// TIA Portal V17 export
// export: Created 2025-06-25T13:13:12.3552397Z, ExportSetting WithDefaults, DisplayName Totally Integrated Automation Portal, DisplayVersion V17 Update 8, DisplayName TIA Portal Openness, DisplayVersion V17 Update 8, DisplayName TIA Portal Version Control Interface, DisplayVersion V17, DisplayName STEP 7 Professional, DisplayVersion V17 Update 8, DisplayName STEP 7 Safety, DisplayVersion V17 Update 6, DisplayName WinCC Advanced, DisplayVersion V17 Update 8
FUNCTION "DigitalOutputProcessing" : Void   // FC11, FBD
TITLE = Output mapping
{ S7_Optimized_Access := 'TRUE' }
VERSION : 0.1
// stored: AutoNumber true, IsIECCheckEnabled false, SetENOAutomatically false, UDAEnableTagReadback false
   VAR_TEMP
      Spare : Bool;
   END_VAR
BEGIN

REGION Network 1: Emergency Stop output
   // 1 = ok, 0 = emergency stop
   // If emergency stop is not active, or you want to reset the safety relay, output is high.
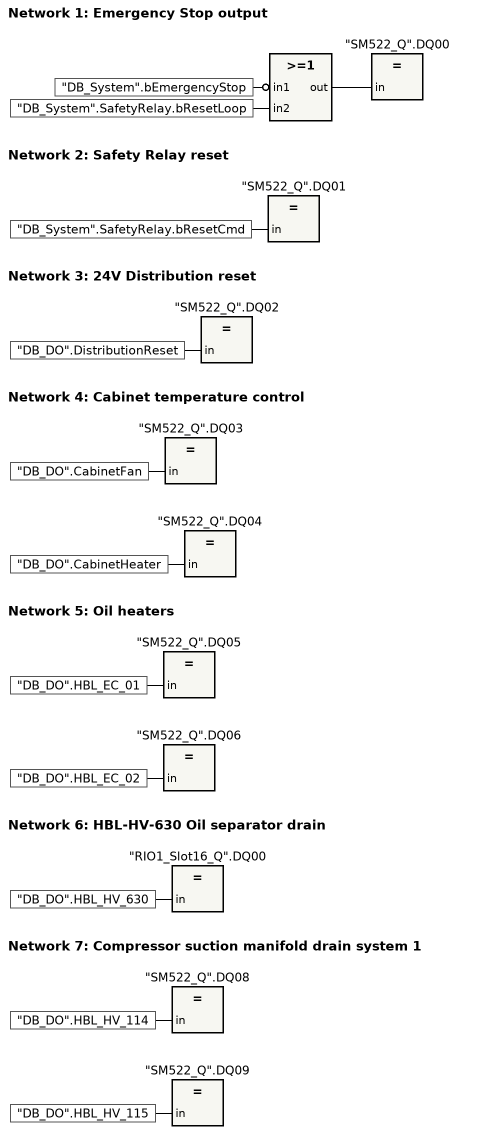
   "SM522_Q".DQ00 := NOT "DB_System".bEmergencyStop OR "DB_System".SafetyRelay.bResetLoop;
END_REGION

REGION Network 2: Safety Relay reset
   "SM522_Q".DQ01 := "DB_System".SafetyRelay.bResetCmd;
END_REGION

REGION Network 3: 24V Distribution reset
   "SM522_Q".DQ02 := "DB_DO".DistributionReset;
END_REGION

REGION Network 4: Cabinet temperature control
   "SM522_Q".DQ03 := "DB_DO".CabinetFan;
   "SM522_Q".DQ04 := "DB_DO".CabinetHeater;
END_REGION

REGION Network 5: Oil heaters
   "SM522_Q".DQ05 := "DB_DO".HBL_EC_01;
   "SM522_Q".DQ06 := "DB_DO".HBL_EC_02;
END_REGION

REGION Network 6: HBL-HV-630 Oil separator drain
   "RIO1_Slot16_Q".DQ00 := "DB_DO".HBL_HV_630;
END_REGION

REGION Network 7: Compressor suction manifold drain system 1
   // Valves directly from suction manifold to sump (optional)
   "SM522_Q".DQ08 := "DB_DO".HBL_HV_114;
   "SM522_Q".DQ09 := "DB_DO".HBL_HV_115;
END_REGION

REGION Network 8: Shaft Seal Cartridge (SSC)
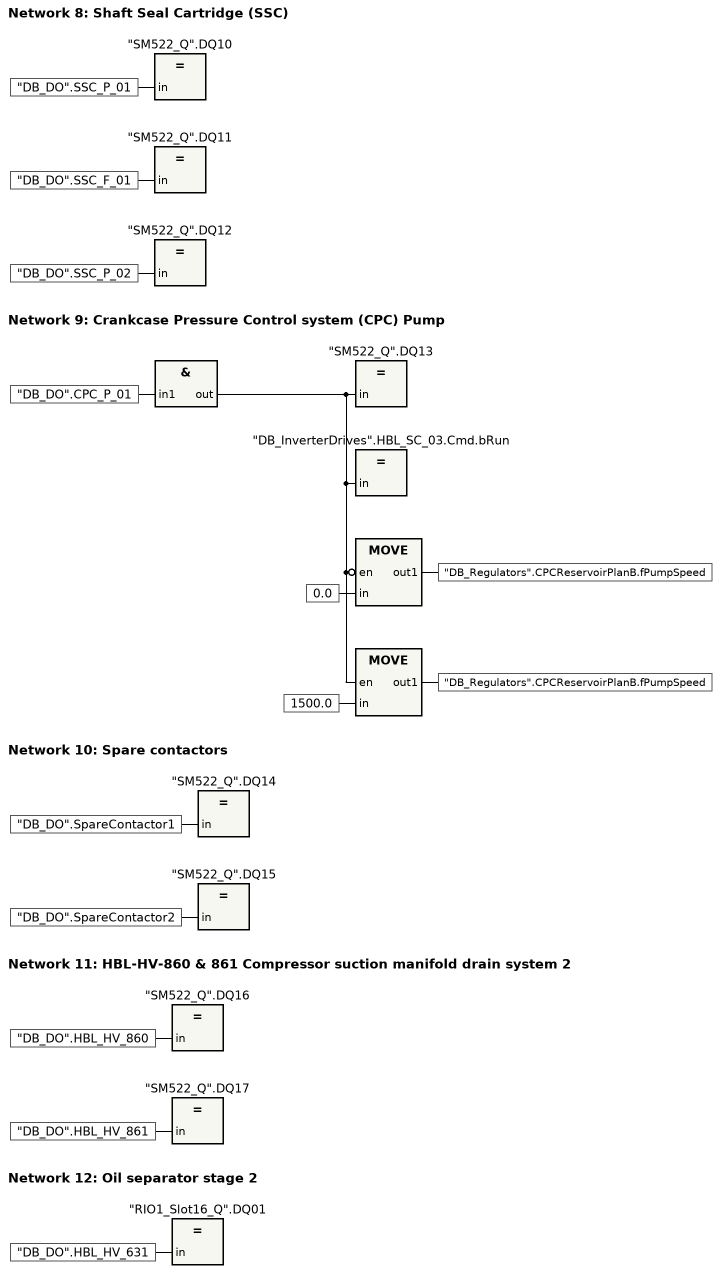
   "SM522_Q".DQ10 := "DB_DO".SSC_P_01;
   "SM522_Q".DQ11 := "DB_DO".SSC_F_01;
   "SM522_Q".DQ12 := "DB_DO".SSC_P_02;
END_REGION

REGION Network 9: Crankcase Pressure Control system (CPC) Pump
   // 10.02.2025 TSS: Normally DQ13, but now an inverter. And this is the ugly hack to make it work until we know how it really should be.
   "SM522_Q".DQ13 := "DB_DO".CPC_P_01;
   "DB_InverterDrives".HBL_SC_03.Cmd.bRun := "DB_DO".CPC_P_01;
   IF NOT "DB_DO".CPC_P_01 THEN "DB_Regulators".CPCReservoirPlanB.fPumpSpeed := 0.0; END_IF;
   IF "DB_DO".CPC_P_01 THEN "DB_Regulators".CPCReservoirPlanB.fPumpSpeed := 1500.0; END_IF;
END_REGION

REGION Network 10: Spare contactors
   "SM522_Q".DQ14 := "DB_DO".SpareContactor1;
   "SM522_Q".DQ15 := "DB_DO".SpareContactor2;
END_REGION

REGION Network 11: HBL-HV-860 & 861 Compressor suction manifold drain system 2
   // Valves to share the CPC system with the Purge controller
   "SM522_Q".DQ16 := "DB_DO".HBL_HV_860;
   "SM522_Q".DQ17 := "DB_DO".HBL_HV_861;
END_REGION

REGION Network 12: Oil separator stage 2
   "RIO1_Slot16_Q".DQ01 := "DB_DO".HBL_HV_631;
END_REGION

REGION Network 13: HBL-HV-640
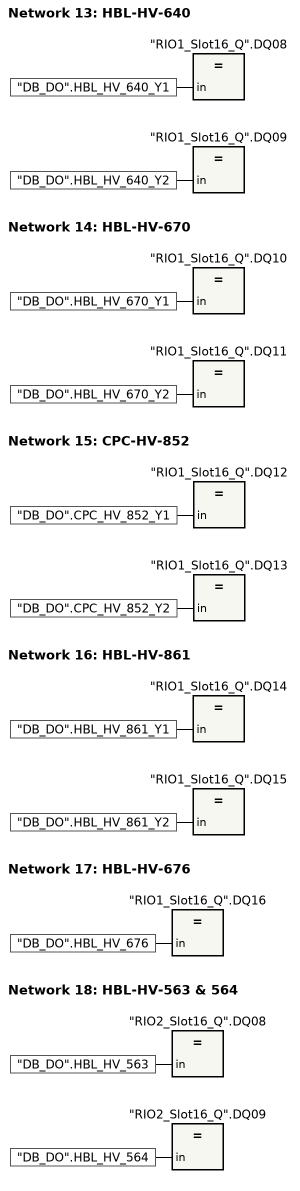
   "RIO1_Slot16_Q".DQ08 := "DB_DO".HBL_HV_640_Y1;
   "RIO1_Slot16_Q".DQ09 := "DB_DO".HBL_HV_640_Y2;
END_REGION

REGION Network 14: HBL-HV-670
   "RIO1_Slot16_Q".DQ10 := "DB_DO".HBL_HV_670_Y1;
   "RIO1_Slot16_Q".DQ11 := "DB_DO".HBL_HV_670_Y2;
END_REGION

REGION Network 15: CPC-HV-852
   "RIO1_Slot16_Q".DQ12 := "DB_DO".CPC_HV_852_Y1;
   "RIO1_Slot16_Q".DQ13 := "DB_DO".CPC_HV_852_Y2;
END_REGION

REGION Network 16: HBL-HV-861
   "RIO1_Slot16_Q".DQ14 := "DB_DO".HBL_HV_861_Y1;
   "RIO1_Slot16_Q".DQ15 := "DB_DO".HBL_HV_861_Y2;
END_REGION

REGION Network 17: HBL-HV-676
   "RIO1_Slot16_Q".DQ16 := "DB_DO".HBL_HV_676;
END_REGION

REGION Network 18: HBL-HV-563 & 564
   "RIO2_Slot16_Q".DQ08 := "DB_DO".HBL_HV_563;
   "RIO2_Slot16_Q".DQ09 := "DB_DO".HBL_HV_564;
END_REGION
END_FUNCTION
